{attribute addProperty BoxType "AMP8000-0000-0103-0103"}
{attribute addProperty Id "Ch_A_AxisMain_InputsCh_A_AxisMain_Inputs_19BB612D648Ch_A_AxisMain_OutputsCh_A_AxisMain_Outputs_1B3A309C162Ch_A_Interpolator_OutputsCh_A_Interpolator_Outputs_70719997648Ch_A_PositionControl_InputsCh_A_PositionControl_Inputs_57B958FE324"}
{attribute addProperty CRC "2977006242"}
{attribute addProperty SizeInBites "176"}
{attribute addProperty SizeInBytes "22"}
TYPE Ch_A_B17182A2 :
STRUCT
	{attribute addProperty Name "Ch_A_AxisMain_Inputs"}
	Ch_A_AxisMain_Inputs  : Ch_A_AxisMain_Inputs_19BB612D;
	{attribute addProperty Name "Ch_A_AxisMain_Outputs"}
	Ch_A_AxisMain_Outputs  : Ch_A_AxisMain_Outputs_1B3A309C;
	{attribute addProperty Name "Ch_A_Interpolator_Outputs"}
	Ch_A_Interpolator_Outputs  : Ch_A_Interpolator_Outputs_70719997;
	{attribute addProperty Name "Ch_A_PositionControl_Inputs"}
	Ch_A_PositionControl_Inputs  : Ch_A_PositionControl_Inputs_57B958FE;
END_STRUCT
END_TYPE

(* stored: Version 1.2.0.0, ProductVersion 3.1.4024.9
   DUT Ch_A_B17182A2: Id {d3fb5dae-d041-4eed-87d6-7891bbc0f6cc} *)
